// TIA Portal V17 export
// export: Created 2024-10-09T16:19:42.5725217Z, ExportSetting WithDefaults, DisplayName Totally Integrated Automation Portal, DisplayVersion V17, DisplayName TIA Portal Openness, DisplayVersion V17, DisplayName TIA Portal Version Control Interface, DisplayVersion V17, DisplayName STEP 7 Professional, DisplayVersion V17, DisplayName STEP 7 Safety, DisplayVersion V17, DisplayName WinCC Advanced, DisplayVersion V17
FUNCTION_BLOCK "ReadWriteControls"   // FB1, LAD
{ S7_Optimized_Access := 'TRUE' }
VERSION : 0.1
// Otomakeit Solutions / 2023
//  -------------------------------------------------------------------------------
//   Title:            ReadWriteControls FB
//   Comment/Function: The Main Control System FB of the project. Collects all inputs from operator controls, outputs operator indication, sets the state of the machine and sends commands to the 
// equipment. 
//                     
//   Library/Family:   LOMS - Master Copies - Project-specific blocks - 20230427_HWDT_AltanticTowing
//   Author:           the Product/Industrial Control Design/Yuriy Mosiyenko
//   Tested with:      1214C, v4.5
//   Engineering:      TIA V17
//   Restrictions:     
//   Requirements:     
//  -------------------------------------------------------------------------------
//   Change log table:
//  Version     | Date             | Expert in charge        | Changes applied
//  ------------------|-----------------------|--------------------------------------|------------------------------
//   00.00.01 | 2023-05-21 | Yuriy Mosiyenko        | Development started
// stored: AutoNumber true, IsIECCheckEnabled true, IsRetainMemResEnabled false, MemoryReserve 100, SetENOAutomatically false, UDAEnableTagReadback false
   VAR_INPUT
      enable { ExternalAccessible := 'False'; ExternalVisible := 'False'; ExternalWritable := 'False'} : Bool;
      mpDI { ExternalAccessible := 'False'; ExternalVisible := 'False'; ExternalWritable := 'False'} : "typeMainPanelDI";   // Main Panel Digital Inputs
      whDI { ExternalAccessible := 'False'; ExternalVisible := 'False'; ExternalWritable := 'False'} : "typeWheelHouseDI";   // Wheel House Digital inputs
      whAI { ExternalAccessible := 'False'; ExternalVisible := 'False'; ExternalWritable := 'False'} : "typeWheelHouseAI";   // Wheel House Analog inputs
      deckDI { ExternalAccessible := 'False'; ExternalVisible := 'False'; ExternalWritable := 'False'} : "typeDeckControlDI";   // Deck Console Digital inputs
      deckAI { ExternalAccessible := 'False'; ExternalVisible := 'False'; ExternalWritable := 'False'} : "typeDeckControlAI";   // Deck Console Analog Inputs
      equipStatus { ExternalAccessible := 'False'; ExternalVisible := 'False'; ExternalWritable := 'False'} : "typeEquipStatus";   // Equipment status feedback
   END_VAR
   VAR_OUTPUT
      alarmWord1 { ExternalVisible := 'False'; ExternalWritable := 'False'} : Word;
      alarmWord2 { ExternalVisible := 'False'; ExternalWritable := 'False'} : Word;
      alarmWord3 { ExternalVisible := 'False'; ExternalWritable := 'False'} : Word;
      shutdownWord { ExternalVisible := 'False'; ExternalWritable := 'False'} : Word;
      mpControlOutputs { ExternalAccessible := 'False'; ExternalVisible := 'False'; ExternalWritable := 'False'} : "typeMpControlOutputs";
      whDQ { ExternalAccessible := 'False'; ExternalVisible := 'False'; ExternalWritable := 'False'} : "typeWheelHouseDQ";   // Wheel House Digital Outputs
      whAQ { ExternalAccessible := 'False'; ExternalVisible := 'False'; ExternalWritable := 'False'} : "typeWheelHouseAQ";   // Wheel House Analog Outputs
      deckDQ { ExternalAccessible := 'False'; ExternalVisible := 'False'; ExternalWritable := 'False'} : "typeDeckControlDQ";   // Deck Console Digital Outputs
      dataToHMI { ExternalAccessible := 'False'; ExternalVisible := 'False'; ExternalWritable := 'False'} : "typeDataToHMI";
      equipCmd : "typeEquipCmd";   // Equipment command data
   END_VAR
   VAR
      statAlarmReset { ExternalAccessible := 'False'; ExternalVisible := 'False'; ExternalWritable := 'False'} : Bool;
      statSafetyStatus { ExternalAccessible := 'False'; ExternalVisible := 'False'; ExternalWritable := 'False'} : Bool;
      statAlarmActive { ExternalAccessible := 'False'; ExternalVisible := 'False'; ExternalWritable := 'False'} : Bool;
      statShutDownActive { ExternalAccessible := 'False'; ExternalVisible := 'False'; ExternalWritable := 'False'} : Bool;
      statAlarmAcknowledged { ExternalAccessible := 'False'; ExternalVisible := 'False'; ExternalWritable := 'False'} : Bool;
      statAlarmWord { ExternalAccessible := 'False'; ExternalVisible := 'False'; ExternalWritable := 'False'} : Word;
      statAlarmWord2 { ExternalAccessible := 'False'; ExternalVisible := 'False'; ExternalWritable := 'False'} : Word;
      statAlarmWord3 { ExternalAccessible := 'False'; ExternalVisible := 'False'; ExternalWritable := 'False'} : Word;
      statShutdownWord { ExternalAccessible := 'False'; ExternalVisible := 'False'; ExternalWritable := 'False'} : Word;
      statDeckCommands { ExternalAccessible := 'False'; ExternalVisible := 'False'; ExternalWritable := 'False'} : "typeDeckStatus";
      statBridgeCommands { ExternalAccessible := 'False'; ExternalVisible := 'False'; ExternalWritable := 'False'; S7_SetPoint := 'True'} : "typeWheelHouseStatus";
      statMpCommands { ExternalAccessible := 'False'; ExternalVisible := 'False'; ExternalWritable := 'False'; S7_SetPoint := 'True'} : "typeMainPanelStatus";
      instReadOperatorControls { ExternalAccessible := 'False'; ExternalVisible := 'False'; ExternalWritable := 'False'; S7_SetPoint := 'True'} : "ReadOperatorControls";
      instSetAlarmsShutdowns { ExternalAccessible := 'False'; ExternalVisible := 'False'; ExternalWritable := 'False'; S7_SetPoint := 'True'} : "SetAlarmsShutdowns";
      instSetMachineState { S7_SetPoint := 'True'} : "SetMachineState";
      instSetResetSafety { ExternalAccessible := 'False'; ExternalVisible := 'False'; ExternalWritable := 'False'; S7_SetPoint := 'True'} : "SetResetSafety";
      instWriteStatusIndicators { S7_SetPoint := 'True'} : "WriteStatusIndicators";
   END_VAR
BEGIN

REGION Network 1: Read Operator Consoles
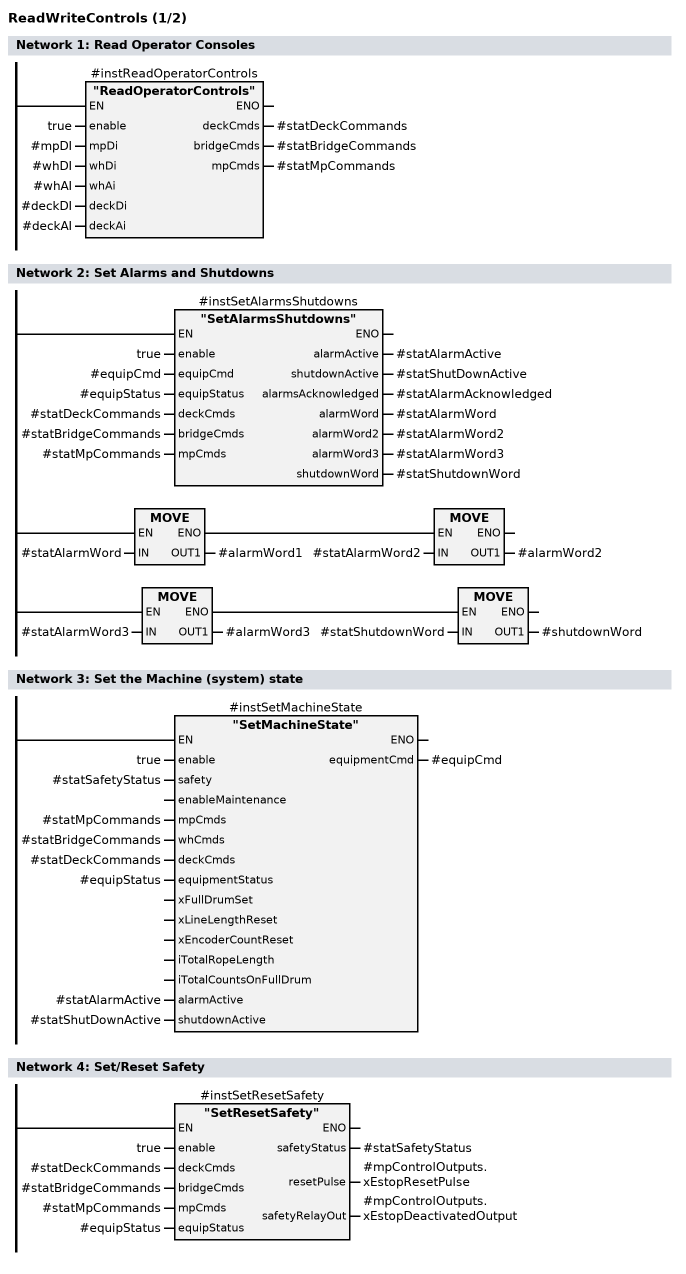
   RUNG wire#powerrail
      #instReadOperatorControls(enable := true, mpDi := #mpDI, whDi := #whDI, whAi := #whAI, deckDi := #deckDI, deckAi := #deckAI, deckCmds => #statDeckCommands, bridgeCmds => #statBridgeCommands, mpCmds => #statMpCommands)
   END_RUNG
   // the same network as SCL:
   #instReadOperatorControls(enable := true,   // "ReadOperatorControls"
                           mpDi := #mpDI,
                           whDi := #whDI,
                           whAi := #whAI,
                           deckDi := #deckDI,
                           deckAi := #deckAI,
                           deckCmds => #statDeckCommands,
                           bridgeCmds => #statBridgeCommands,
                           mpCmds => #statMpCommands);
END_REGION

REGION Network 2: Set Alarms and Shutdowns
   RUNG wire#powerrail
      #instSetAlarmsShutdowns(enable := true, equipCmd := #equipCmd, equipStatus := #equipStatus, deckCmds := #statDeckCommands, bridgeCmds := #statBridgeCommands, mpCmds := #statMpCommands, alarmActive => #statAlarmActive, shutdownActive => #statShutDownActive, alarmsAcknowledged => #statAlarmAcknowledged, alarmWord => #statAlarmWord, alarmWord2 => #statAlarmWord2, alarmWord3 => #statAlarmWord3, shutdownWord => #statShutdownWord)
   END_RUNG
   RUNG wire#powerrail
      Move(in := #statAlarmWord, out1 => #alarmWord1)
      Move(in := #statAlarmWord2, out1 => #alarmWord2)
   END_RUNG
   RUNG wire#powerrail
      Move(in := #statAlarmWord3, out1 => #alarmWord3)
      Move(in := #statShutdownWord, out1 => #shutdownWord)
   END_RUNG
   // the same network as SCL:
   #instSetAlarmsShutdowns(enable := true,   // "SetAlarmsShutdowns"
                           equipCmd := #equipCmd,
                           equipStatus := #equipStatus,
                           deckCmds := #statDeckCommands,
                           bridgeCmds := #statBridgeCommands,
                           mpCmds := #statMpCommands,
                           alarmActive => #statAlarmActive,
                           shutdownActive => #statShutDownActive,
                           alarmsAcknowledged => #statAlarmAcknowledged,
                           alarmWord => #statAlarmWord,
                           alarmWord2 => #statAlarmWord2,
                           alarmWord3 => #statAlarmWord3,
                           shutdownWord => #statShutdownWord);
   #alarmWord1 := #statAlarmWord;
   #alarmWord2 := #statAlarmWord2;
   #alarmWord3 := #statAlarmWord3;
   #shutdownWord := #statShutdownWord;
END_REGION

REGION Network 3: Set the Machine (system) state
   RUNG wire#powerrail
      #instSetMachineState(enable := true, safety := #statSafetyStatus, enableMaintenance :=, mpCmds := #statMpCommands, whCmds := #statBridgeCommands, deckCmds := #statDeckCommands, equipmentStatus := #equipStatus, xFullDrumSet :=, xLineLengthReset :=, xEncoderCountReset :=, iTotalRopeLength :=, iTotalCountsOnFullDrum :=, alarmActive := #statAlarmActive, shutdownActive := #statShutDownActive, equipmentCmd => #equipCmd)
   END_RUNG
   // the same network as SCL:
   #instSetMachineState(enable := true,   // "SetMachineState"
                        safety := #statSafetyStatus,
                        mpCmds := #statMpCommands,
                        whCmds := #statBridgeCommands,
                        deckCmds := #statDeckCommands,
                        equipmentStatus := #equipStatus,
                        alarmActive := #statAlarmActive,
                        shutdownActive := #statShutDownActive,
                        equipmentCmd => #equipCmd);
END_REGION

REGION Network 4: Set/Reset Safety
   RUNG wire#powerrail
      #instSetResetSafety(enable := true, deckCmds := #statDeckCommands, bridgeCmds := #statBridgeCommands, mpCmds := #statMpCommands, equipStatus := #equipStatus, safetyStatus => #statSafetyStatus, resetPulse => #mpControlOutputs.xEstopResetPulse, safetyRelayOut => #mpControlOutputs.xEstopDeactivatedOutput)
   END_RUNG
   // the same network as SCL:
   #instSetResetSafety(enable := true,   // "SetResetSafety"
                       deckCmds := #statDeckCommands,
                       bridgeCmds := #statBridgeCommands,
                       mpCmds := #statMpCommands,
                       equipStatus := #equipStatus,
                       safetyStatus => #statSafetyStatus,
                       resetPulse => #mpControlOutputs.xEstopResetPulse,
                       safetyRelayOut => #mpControlOutputs.xEstopDeactivatedOutput);
END_REGION

REGION Network 5: Output consoles indicators
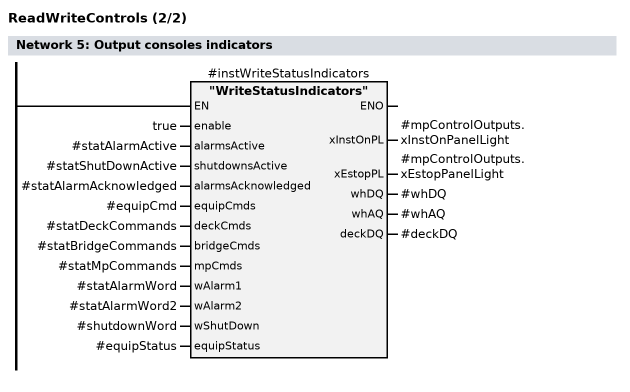
   RUNG wire#powerrail
      #instWriteStatusIndicators(enable := true, alarmsActive := #statAlarmActive, shutdownsActive := #statShutDownActive, alarmsAcknowledged := #statAlarmAcknowledged, equipCmds := #equipCmd, deckCmds := #statDeckCommands, bridgeCmds := #statBridgeCommands, mpCmds := #statMpCommands, wAlarm1 := #statAlarmWord, wAlarm2 := #statAlarmWord2, wShutDown := #shutdownWord, equipStatus := #equipStatus, xInstOnPL => #mpControlOutputs.xInstOnPanelLight, xEstopPL => #mpControlOutputs.xEstopPanelLight, whDQ => #whDQ, whAQ => #whAQ, deckDQ => #deckDQ)
   END_RUNG
   // the same network as SCL:
   #instWriteStatusIndicators(enable := true,   // "WriteStatusIndicators"
                           alarmsActive := #statAlarmActive,
                           shutdownsActive := #statShutDownActive,
                           alarmsAcknowledged := #statAlarmAcknowledged,
                           equipCmds := #equipCmd,
                           deckCmds := #statDeckCommands,
                           bridgeCmds := #statBridgeCommands,
                           mpCmds := #statMpCommands,
                           wAlarm1 := #statAlarmWord,
                           wAlarm2 := #statAlarmWord2,
                           wShutDown := #shutdownWord,
                           equipStatus := #equipStatus,
                           xInstOnPL => #mpControlOutputs.xInstOnPanelLight,
                           xEstopPL => #mpControlOutputs.xEstopPanelLight,
                           whDQ => #whDQ,
                           whAQ => #whAQ,
                           deckDQ => #deckDQ);
END_REGION
END_FUNCTION_BLOCK
